Universal Robots PolyScope program: Lab_exe_5_2_99.urp

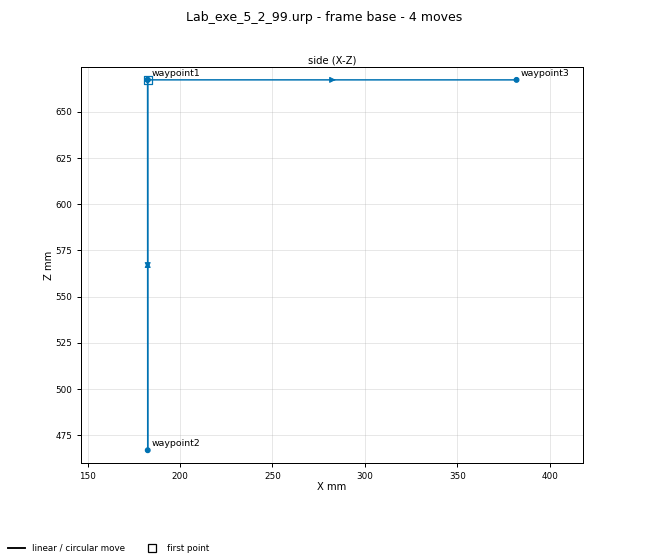
[picture p0: tool path of Lab_exe_5_2_99.urp in frame base, 4 of 4 moves have a stored position in this frame; points joined in program order, loops and branches not executed]
Program Lab_exe_5_2_99 (createdIn=3.2.19293 lastSavedIn=3.2.19293 directory=/programs installation=default robotSerialNumber=2015351391)
Calibrated DH parameters: a=[0.000352, -0.161198, -0.373486, 0.00005, 0.000049, 0]; d=[0.089268, 352.477598, -320.08558, -32.281492, 0.094939, 0.082518]; alpha=[1.570728, 0.001116, -0.003686, 1.571189, -1.570572, 0]; deltaTheta=[-0.000012, 1.181849, -1.491165, 0.309495, -0.000007, 0.000025]
Robot Program (runOnlyOnce=false motionType=MoveJ speed=1.047198 acceleration=1.396263 recalculateMotions=false)
  MoveL speed 250 mm/s, acceleration 1200 mm/s^2 (recalculateMotions=false) feature=Base
    Waypoint waypoint1: TCP in base x=182.482 y=236.698 z=667.301 mm, rx=-1.585 ry=-0.1094 rz=-0.2822 rad; joints [70.438, -65.349, -100.16, -15.213, 103.17, -14.698] deg
    Wait DigitalInput pin=Button; digitalValue=1
    Call SubP_lamp_flash
    Waypoint waypoint2: TCP in base x=182.52 y=236.701 z=466.953 mm, rx=-1.5851 ry=-0.1092 rz=-0.2823 rad; joints [70.361, -65.589, -129.636, 14.507, 103.347, -14.669] deg; flange x=182.495 y=236.694 z=467 mm, rx=-1.585 ry=-0.1094 rz=-0.2823 rad
    If Button≟ True
      Waypoint waypoint1: TCP in base x=182.482 y=236.698 z=667.301 mm, rx=-1.585 ry=-0.1094 rz=-0.2822 rad; joints [70.438, -65.349, -100.16, -15.213, 103.17, -14.698] deg
    Else 
      Waypoint waypoint3: TCP in base x=382.005 y=236.721 z=667.282 mm, rx=-1.5851 ry=-0.1095 rz=-0.2824 rad; joints [38.59, -89.754, -81.535, -9.878, 135.061, -15.288] deg
SubProgram -> SubP_lamp_flash
SubProgram SubP_lamp_flash (keepSynchronizedWithDisk=false trackProgramExecution=false) programFile=/programs/lamp_flash.urp
  Set DigitalOutput pin=Lamp; digitalValue=1
  Wait Sleep waitTime=0.5
  Set DigitalOutput pin=Lamp; digitalValue=0
  Wait Sleep waitTime=0.5
